(* IEC 61131-3 sources: Lasal/CPU_5344_V01/Class/logger, 1 file *)

(* ---- logger.st ---- *)
(*!
<Class
	Name               = "logger"
	Revision           = "0.0"
	RealtimeTask       = "true"
	DefRealtime        = "5 ms"
	CyclicTask         = "false"
	BackgroundTask     = "false"
	Sigmatek           = "false"
	OSInterface        = "false"
	HighPriority       = "false"
	Automatic          = "false"
	UpdateMode         = "Prescan"
	SharedCommandTable = "true"
	Objectsize         = "(284,120)">
	<Channels>
		<Server Name="close" Visualized="false" Initialize="false" WriteProtected="false" Retentive="false"/>
		<Server Name="open" Visualized="false" Initialize="false" WriteProtected="false" Retentive="false"/>
		<Server Name="writeLine" Visualized="false" Initialize="false" WriteProtected="false" Retentive="false"/>
		<Client Name="fileBase" Required="true" Internal="false"/>
		<Client Name="fileSys" Required="false" Internal="false"/>
		<Client Name="minValue" Required="true" Internal="false"/>
		<Client Name="value1" Required="true" Internal="false"/>
		<Client Name="value2" Required="true" Internal="false"/>
		<Client Name="value3" Required="true" Internal="false"/>
	</Channels>
</Class>
*)
logger : CLASS
  //Servers:
	open 	: SvrChCmd_DINT;
	writeLine 	: SvrCh_DINT;
	close 	: SvrCh_DINT;
  //Clients:
	fileSys 	: CltChCmd__FileSys;
	fileBase 	: CltChCmd_FileBase;
	minValue 	: CltCh_DINT;
	value1 	: CltCh_DINT;
	value2 	: CltCh_DINT;
	value3 	: CltCh_DINT;
  //Variables:
		handle 	: DINT;
		string : ARRAY [0..100] OF CHAR;

		len 	: DINT;
  //Functions:

	FUNCTION VIRTUAL GLOBAL RtWork
		VAR_INPUT
			EAX 	: UDINT;
		END_VAR
		VAR_OUTPUT
			state (EAX) 	: UDINT := READY;
		END_VAR;

	FUNCTION VIRTUAL GLOBAL open::Write
		VAR_INPUT
			input (EAX) 	: DINT;
		END_VAR
		VAR_OUTPUT
			result (EAX) 	: DINT;
		END_VAR;

	FUNCTION VIRTUAL GLOBAL writeLine::Write
		VAR_INPUT
			input (EAX) 	: DINT;
		END_VAR
		VAR_OUTPUT
			result (EAX) 	: DINT;
		END_VAR;

	FUNCTION VIRTUAL GLOBAL close::Write
		VAR_INPUT
			input (EAX) 	: DINT;
		END_VAR
		VAR_OUTPUT
			result (EAX) 	: DINT;
		END_VAR;
  //Tables:
	FUNCTION @STD
		VAR_OUTPUT
			ret_code	: CONFSTATES;
		END_VAR;
	FUNCTION GLOBAL TAB @CT_;
END_CLASS;

#pragma usingLtd _FileSys
#pragma usingLtd FileBase

FUNCTION VIRTUAL GLOBAL logger::open::Write
	VAR_INPUT
		input (EAX) 	: DINT;
	END_VAR
	VAR_OUTPUT
		result (EAX) 	: DINT;
	END_VAR

	open := input;

  handle:=fileSys.FileOpen(filename:="c:\file.csv", attributes:=ATT_CREATE);
  close:=0;

	result := open;

END_FUNCTION

FUNCTION VIRTUAL GLOBAL logger::writeLine::Write
	VAR_INPUT
		input (EAX) 	: DINT;
	END_VAR
	VAR_OUTPUT
		result (EAX) 	: DINT;
	END_VAR

	writeLine := input;
  IF handle > 0 THEN
    writeline:= fileSys.FileWrite(handle:=handle, buffer:=#string[0], length:=_strlen(src:=#string[0]));

  END_IF;
	result := writeLine;

END_FUNCTION

FUNCTION VIRTUAL GLOBAL logger::close::Write
	VAR_INPUT
		input (EAX) 	: DINT;
	END_VAR
	VAR_OUTPUT
		result (EAX) 	: DINT;
	END_VAR

	close := input;
  IF handle > 0 THEN
    fileSys.FileClose(handle:=handle);
  END_IF;
	result := close;

END_FUNCTION

FUNCTION VIRTUAL GLOBAL logger::RtWork
	VAR_INPUT
		EAX 	: UDINT;
	END_VAR
	VAR_OUTPUT
		state (EAX) 	: UDINT;(* := READY *)
	END_VAR

  minValue:=minValue.Read();

  IF handle> 0 & close= 0 & minValue>=23 & minValue<= 27 THEN
    value1 := value1.Read();
    value2 := value2.Read();
    value3 := value3.Read();

    _memset(dest:=#string[0], usByte:=0, cntr:=sizeof(string));

    fileBase.BuildValue2Ascii(Value:=value1, Dest:=#string[0], Offset:=0);
    len:=to_dint(_strlen(src:=#string[0]));
    string[len]:=';';
    fileBase.BuildValue2Ascii(Value:=value2, Dest:=#string[len+1], Offset:=0);
    len:=to_dint(_strlen(src:=#string[0]));
    string[len]:=';';
    fileBase.BuildValue2Ascii(Value:=value3, Dest:=#string[len+1], Offset:=0);
    len:=to_dint(_strlen(src:=#string[0]));
    string[len]:=13;

    fileSys.FileWrite(handle:=handle, buffer:=#string[0], length:=_strlen(src:=#string[0]));

  END_IF;

END_FUNCTION
